// TIA Portal V19 export
// export: Created 2019-11-11T12:29:20.5206584Z, ExportSetting None
DATA_BLOCK "DriveLogic_DB"   // DB4
{ S7_Optimized_Access := 'TRUE' }
// stored: InstanceOfName DriveLogic, InstanceOfType FB
"DriveLogic"
   // VAR_INPUT
   //    Enable_Drives : Bool;
   //    AckError : Bool;
   //    SpeedSp : Real;
   // END_VAR
   // VAR
   //    SINA_SPEED_Instance_1 { S7_SetPoint := 'True'} : "SINA_SPEED";
   // END_VAR
BEGIN
END_DATA_BLOCK
